// TIA Portal V17 export
// export: Created 2024-06-16T17:47:27.1808862Z, ExportSetting WithDefaults, DisplayName Totally Integrated Automation Portal, DisplayVersion V17, DisplayName TIA Portal Openness, DisplayVersion V17, DisplayName TIA Portal Version Control Interface, DisplayVersion V17, DisplayName STEP 7 Professional, DisplayVersion V17, DisplayName STEP 7 Safety, DisplayVersion V17, DisplayName WinCC Professional, DisplayVersion V17
FUNCTION_BLOCK "Obj_St2_FB"   // FB200, FBD
{ S7_Optimized_Access := 'TRUE' }
VERSION : 0.1
// stored: AutoNumber false, IsIECCheckEnabled false, IsRetainMemResEnabled false, MemoryReserve 100, SetENOAutomatically false, UDAEnableTagReadback false
   VAR
      Axe_X1 : Struct
         _ActPos : Real;
         _ActVel : Real;
         _Mode : Int;
         Home : Bool;
         Halt : Bool;
         Jog : Bool;
         MoveAbs : Bool;
         MoveRel : Bool;
         MoveVel : Bool;
         PowerOff : Bool;
         PowerOn : Bool;
         SensPos : Bool;
         SensNeg : Bool;
         xBusy : Bool;
         xHomed : Bool;
         xMoveAbsDone : Bool;
         xMoveRelDone : Bool;
         xPower : Bool;
      END_STRUCT;
      Axe_X2 : Struct
         _ActPos : Real;
         _ActVel : Real;
         _Mode : Int;
         Home : Bool;
         Halt : Bool;
         Jog : Bool;
         MoveAbs : Bool;
         MoveRel : Bool;
         MoveVel : Bool;
         PowerOff : Bool;
         PowerOn : Bool;
         SensPos : Bool;
         SensNeg : Bool;
         xBusy : Bool;
         xHomed : Bool;
         xMoveAbsDone : Bool;
         xMoveRelDone : Bool;
         xPower : Bool;
      END_STRUCT;
      Prehenseur_Z : Struct
         _ActPos : Real;
         _ActVel : Real;
         _Mode : Int;
         Home : Bool;
         Halt : Bool;
         Jog : Bool;
         MoveAbs : Bool;
         MoveRel : Bool;
         MoveVel : Bool;
         PowerOff : Bool;
         PowerOn : Bool;
         SensPos : Bool;
         SensNeg : Bool;
         xBusy : Bool;
         xHomed : Bool;
         xMoveAbsDone : Bool;
         xMoveRelDone : Bool;
         xPower : Bool;
      END_STRUCT;
   END_VAR
BEGIN

REGION Network 1: Station 2 - Axe X1
   // //___ ModePose : 
   //          1 ---> Relative positioning
   //          2 ---> Absolute positioning
   //          3 ---> Not supported
   //          4 ---> Referencing - referencing point approach
   //          5 ---> Referencing - set referencing point
   //          6 ---> Traversing block (record mode)
   //          7 ---> Jog
   //          8 ---> Not supported
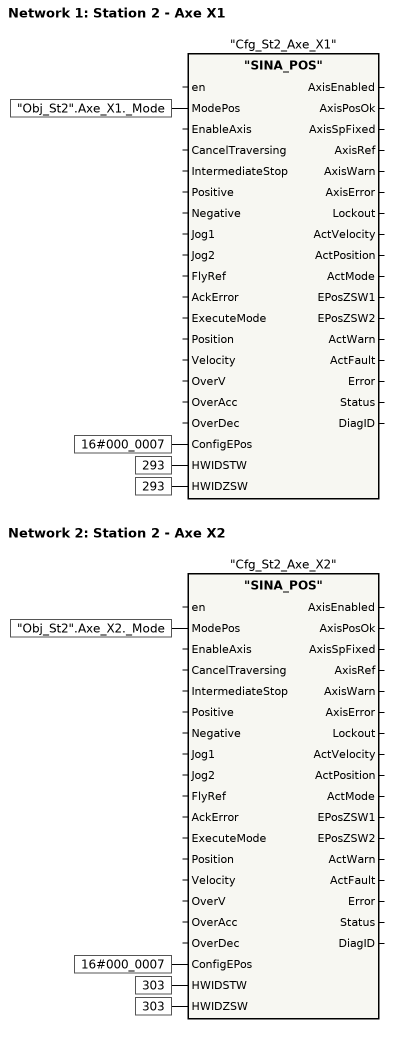
   "Cfg_St2_Axe_X1"(ModePos := "Obj_St2".Axe_X1._Mode,   // "SINA_POS"
                    ConfigEPos := 16#000_0007,
                    HWIDSTW := 293,
                    HWIDZSW := 293);
END_REGION

REGION Network 2: Station 2 - Axe X2
   // //___ ModePose : 
   //          1 ---> Relative positioning
   //          2 ---> Absolute positioning
   //          3 ---> Not supported
   //          4 ---> Referencing - referencing point approach
   //          5 ---> Referencing - set referencing point
   //          6 ---> Traversing block (record mode)
   //          7 ---> Jog
   //          8 ---> Not supported
   "Cfg_St2_Axe_X2"(ModePos := "Obj_St2".Axe_X2._Mode,   // "SINA_POS"
                    ConfigEPos := 16#000_0007,
                    HWIDSTW := 303,
                    HWIDZSW := 303);
END_REGION

REGION Network 3: Station 2 - Prehenseur Z
   // //___ ModePose : 
   //          1 ---> Relative positioning
   //          2 ---> Absolute positioning
   //          3 ---> Not supported
   //          4 ---> Referencing - referencing point approach
   //          5 ---> Referencing - set referencing point
   //          6 ---> Traversing block (record mode)
   //          7 ---> Jog
   //          8 ---> Not supported
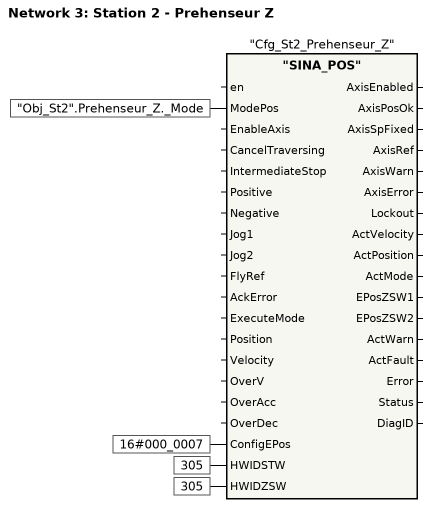
   "Cfg_St2_Prehenseur_Z"(ModePos := "Obj_St2".Prehenseur_Z._Mode,   // "SINA_POS"
                          ConfigEPos := 16#000_0007,
                          HWIDSTW := 305,
                          HWIDZSW := 305);
END_REGION
END_FUNCTION_BLOCK
